// TIA Portal V20 export
DATA_BLOCK "Com_DB"   // DB301
// stored: AutoNumber false, InstanceOfName Com, InstanceOfType FB
"Com"
   // VAR
   //    Var { S7_SetPoint := 'True'} : "TypeVar";
   //    T : Array[1..6] of IEC_TIMER;
   //    wdOldParam { ExternalAccessible := 'False'; ExternalVisible := 'False'; ExternalWritable := 'False'} : Int;
   //    wdOldErr { ExternalAccessible := 'False'; ExternalVisible := 'False'; ExternalWritable := 'False'} : Int;
   // END_VAR
BEGIN
END_DATA_BLOCK
